FUNCTION_BLOCK FB_MoveStepperLoop
VAR_INPUT
	stepsToMove				: INT;
	PosCurrent				: UDINT;
END_VAR
VAR_OUTPUT
END_VAR
VAR
	Step 					: INT := 0;
	bPowerOn				: INT;
END_VAR

MAIN.fbAxis1.bEnable := TRUE;

CASE Step OF
0:
	MAIN.fbAxis1.moveRelDist := 0.0;
	MAIN.fbAxis1.moveRelVel := 0.0;
	MAIN.fbAxis1.bMoveRelExe := FALSE;
	MAIN.fbAxis1.bHaltExe := FALSE;
	Step := 1;
1:

	IF MAIN.fbAxis1.bPwrStatus THEN
		MAIN.fbAxis1.moveRelDist := 1;
		MAIN.fbAxis1.moveRelVel := 100;
		MAIN.fbAxis1.bMoveRelExe := TRUE;
		IF MAIN.fbAxis1.bMoveRelDone THEN
			MAIN.fbAxis1.bMoveRelExe := FALSE;
			MAIN.fbAxis1.bHaltExe := TRUE;
		END_IF
	END_IF
	StepsToMove := StepsToMove - 1;
	Step := 2;
2:
	IF MAIN.fbAxis1.bHaltDone = TRUE THEN
		MAIN.fbAxis1.bHaltExe := FALSE;
	END_IF

	MAIN.bMoveRelative := FALSE;
	IF StepsToMove = 0 THEN
		Step := 3;
	ELSE
		Step := 0;
	END_IF
END_CASE

END_FUNCTION_BLOCK

(* stored: Version 1.1.0.1, ProductVersion 3.1.4024.9
   POU FB_MoveStepperLoop: Id {94a3cc5b-b61b-4cf3-a90b-6edb0ed7f1c8}, SpecialFunc None *)
